FUNCTION_BLOCK WaterMonitor_HCECC
  (* Standard: 61499-2 *)
  (* Version 0.2, 2003-12-05, JHC, Rockwell Automation, Renamed from NEWCOMPFB. *)
  (* Compiler header: package fb.rt.benchmarks.watermonitor; *)
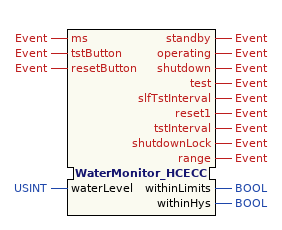
  EVENT_INPUT
    ms; (* millisecond *)
    tstButton;
    resetButton;
  END_EVENT
  EVENT_OUTPUT
    standby;
    operating;
    shutdown;
    test;
    slfTstInterval;
    reset1;
    tstInterval;
    shutdownLock;
    range;
  END_EVENT
  VAR_INPUT
    waterLevel : USINT;
  END_VAR
  VAR_OUTPUT
    withinLimits : BOOL;
    withinHys : BOOL;
  END_VAR
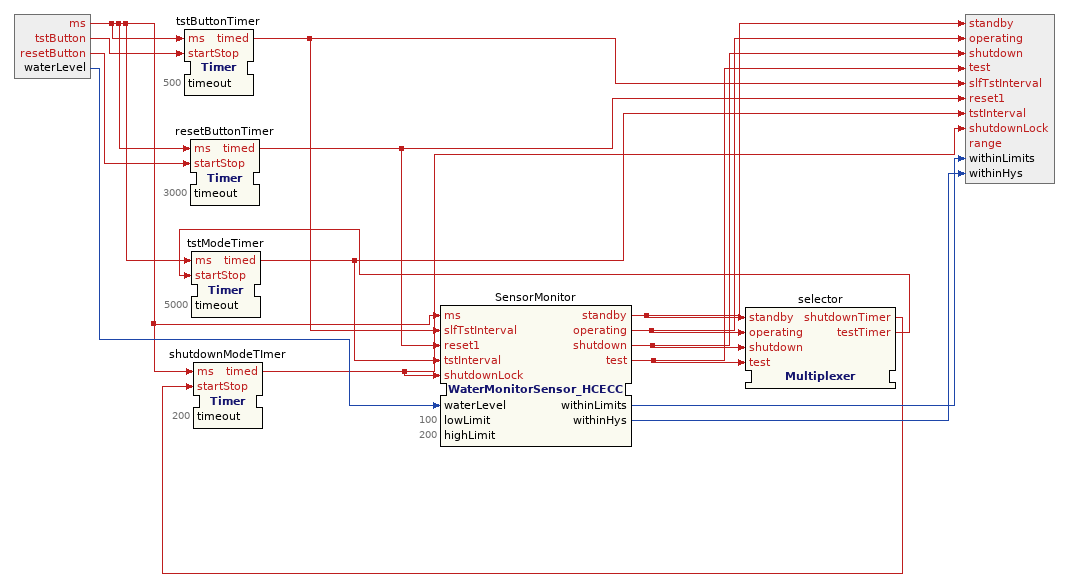
  FBS
    SensorMonitor : WaterMonitorSensor_HCECC(lowLimit := 100, highLimit := 200);
    tstButtonTimer : Timer(timeout := 500);
    tstModeTimer : Timer(timeout := 5000);
    shutdownModeTImer : Timer(timeout := 200);
    resetButtonTimer : Timer(timeout := 3000);
    selector : Multiplexer;
  END_FBS
  EVENT_CONNECTIONS
    ms TO SensorMonitor.ms;
    ms TO tstButtonTimer.ms;
    ms TO resetButtonTimer.ms;
    ms TO tstModeTimer.ms;
    tstButton TO tstButtonTimer.startStop;
    resetButton TO resetButtonTimer.startStop;
    tstButtonTimer.timed TO SensorMonitor.slfTstInterval;
    resetButtonTimer.timed TO SensorMonitor.reset1;
    tstModeTimer.timed TO SensorMonitor.tstInterval;
    shutdownModeTImer.timed TO SensorMonitor.shutdownLock;
    ms TO shutdownModeTImer.ms;
    SensorMonitor.standby TO selector.standby;
    SensorMonitor.operating TO selector.operating;
    SensorMonitor.shutdown TO selector.shutdown;
    SensorMonitor.test TO selector.test;
    selector.shutdownTimer TO shutdownModeTImer.startStop;
    selector.testTimer TO tstModeTimer.startStop;
    SensorMonitor.standby TO standby;
    SensorMonitor.operating TO operating;
    SensorMonitor.shutdown TO shutdown;
    SensorMonitor.test TO test;
    tstButtonTimer.timed TO slfTstInterval;
    tstModeTimer.timed TO tstInterval;
    resetButtonTimer.timed TO reset1;
    shutdownModeTImer.timed TO shutdownLock;
  END_CONNECTIONS
  DATA_CONNECTIONS
    waterLevel TO SensorMonitor.waterLevel;
    SensorMonitor.withinLimits TO withinLimits;
    SensorMonitor.withinHys TO withinHys;
  END_CONNECTIONS
END_FUNCTION_BLOCK
